// TIA Portal V20 export
ORGANIZATION_BLOCK "Main"   // OB1001, LAD, ProgramCycle
TITLE = "Main Program Sweep (Cycle)"
// This block calls the FB CallUnit which includes all further functionality of the unit.
// It reads the general global status and the safety status from the respective safety zone.
// It writes the unit status back to the DB Global.Data and the acknowledge information to the respetive safety zone.
// OB Main is a program cycle OB and is called depending on its number. For details, refer to the Automation Framework documentation.
// stored: AutoNumber false, IsIECCheckEnabled true, Namespace Unit1, SetENOAutomatically true
   VAR_INPUT
      Initial_Call : Bool;   // Initial call of this OB
      Remanence : Bool;   // =True, if remanent data are available
   END_VAR
   VAR_TEMP
      tempIndex : Int;   // Index of Unit in the array
      tempStart : Bool;
   END_VAR
   VAR CONSTANT
      "Temporary bit" : Bool := true;
      AlwaysTrue : Bool := true;
   END_VAR
BEGIN

REGION Network 1: System Stable time
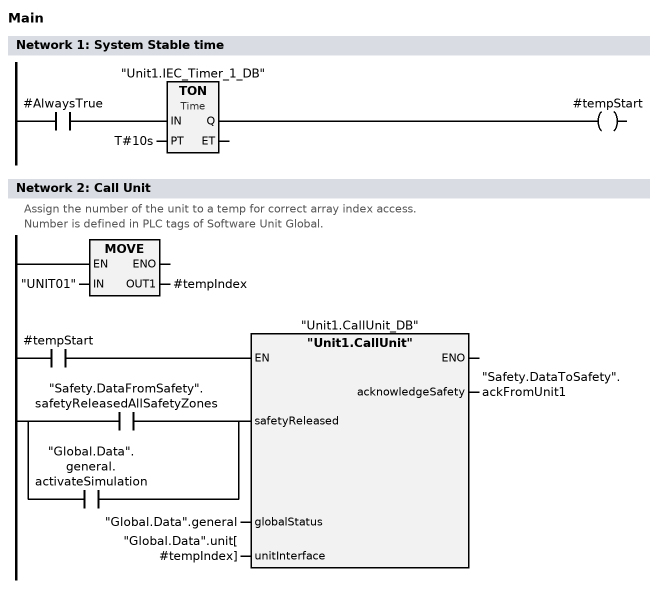
   RUNG wire#powerrail
      Contact( #AlwaysTrue )
      { S7_Templates := "time_type := Time" } "Unit1.IEC_Timer_1_DB".TON(pt := T#10s, et =>)
      Coil( #tempStart )
   END_RUNG
   // the same network as SCL:
   "Unit1.IEC_Timer_1_DB".TON(IN := #AlwaysTrue, PT := T#10s);
   #tempStart := "Unit1.IEC_Timer_1_DB".Q;
END_REGION

REGION Network 2: Call Unit
   // Assign the number of the unit to a temp for correct array index access.
   // Number is defined in PLC tags of Software Unit Global.
   RUNG wire#powerrail
      Move(in := "UNIT01", out1 => #tempIndex)
   END_RUNG
   RUNG wire#powerrail
      Contact( #tempStart )
      "Unit1.CallUnit_DB"(safetyReleased := wire#w1, globalStatus := "Global.Data".general, unitInterface := "Global.Data".unit[#tempIndex], acknowledgeSafety => "Safety.DataToSafety".ackFromUnit1)
   END_RUNG
   RUNG wire#powerrail
      Contact( "Safety.DataFromSafety".safetyReleasedAllSafetyZones )
   END_RUNG wire#w1
   RUNG wire#powerrail
      Contact( "Global.Data".general.activateSimulation )
   END_RUNG wire#w1
   // the same network as SCL:
   #tempIndex := "UNIT01";
   IF #tempStart THEN
       "Unit1.CallUnit_DB"(safetyReleased := "Safety.DataFromSafety".safetyReleasedAllSafetyZones OR "Global.Data".general.activateSimulation,   // "Unit1.CallUnit"
                           globalStatus := "Global.Data".general,
                           unitInterface := "Global.Data".unit[#tempIndex],
                           acknowledgeSafety => "Safety.DataToSafety".ackFromUnit1);
   END_IF;
END_REGION
END_ORGANIZATION_BLOCK
